FUNCTION_BLOCK BoolPub EXTENDS Object IMPLEMENTS I_BoolSub
VAR_INPUT
	IN: BOOL;
END_VAR
VAR
	_sub: I_BoolSub;
END_VAR

//Work in progress

METHOD Attach_Sub
VAR_INPUT
	IObject: I_SYS_COMP_Object;
END_VAR
VAR
	_ISub: I_BoolSub;
END_VAR
IF __QUERYINTERFACE(IObject, _ISub) THEN
	_sub := _ISub;
END_IF
END_METHOD

PROPERTY Get : I_SYS_COMP_Object
GET
IN := Get;
END_GET
END_PROPERTY

METHOD Remove_Sub
VAR_INPUT
	IObject: I_SYS_COMP_Object;
END_VAR
VAR
	_ISub: I_BoolSub;
END_VAR
IF __QUERYINTERFACE(IObject, _ISub) THEN
	_sub := _ISub;
END_IF
END_METHOD

END_FUNCTION_BLOCK

(* stored: Version 1.1.0.1, ProductVersion 3.1.4024.12
   POU BoolPub: Id {a9a66cfb-679c-4177-804d-f1017675d0b2}, SpecialFunc None
   Method Attach_Sub: Id {b77e8169-6f7d-4619-a088-a9d809e4fcc2}
   Property Get: Id {fc7afd35-76d3-4822-a75b-49ce5b51e532}
   Get Get: Id {074db2a4-4981-4300-9123-fa45daf3dd83}
   Method Remove_Sub: Id {a69b7383-0a35-431f-a75f-7ddf957bd782} *)
